{attribute 'linkalways'} 
{attribute 'no_explicit_call' := 'This FB is a CLASS and must be accessed using methods or properties'}
{attribute 'enable_dynamic_creation'}
FUNCTION_BLOCK FINAL GE_LREAL EXTENDS Node
VAR
	in1 : _LREAL(0.0);
	in2 : _LREAL(0.0);
	out : _BOOL(FALSE);
END_VAR

METHOD PUBLIC Clone : I_Node
VAR
	pNode : POINTER TO GE_LREAL;
END_VAR
pNode := __NEW(GE_LREAL);
Clone := pNode^;
END_METHOD

METHOD FB_init : BOOL
VAR_INPUT
	bInitRetains : BOOL; // if TRUE, the retain variables are initialized (warm start / cold start)
	bInCopyCode : BOOL;  // if TRUE, the instance afterwards gets moved into the copy code (online change)
END_VAR
AddInput('in1',THIS^.in1);
AddInput('in2',THIS^.in2);
AddOutput('out', THIS^.out);
END_METHOD

METHOD PROTECTED OnExecute
VAR
END_VAR
out.Value := in1.Value >= in2.Value;
END_METHOD

END_FUNCTION_BLOCK

(* stored: Version 1.1.0.1, ProductVersion 3.1.4024.15
   POU GE_LREAL: Id {c44a56a5-c7eb-4254-8575-4524d73d08ad}, SpecialFunc None
   Folder Constructor: Id {45563143-99db-497d-9dd3-2e02a88306d2}
   Method Clone: Id {1b328468-e195-45a8-a531-e8737d355afd}
   Method FB_init: Id {eb2bdf1e-9035-4c7e-a7a6-41f1663edd6e}
   Method OnExecute: Id {1f5d5cac-59dc-4223-b502-51b2d8ebb6c2} *)
